Omron CX-Programmer project New_Project (CX-Programmer 9.73)

# PLC NewPLC1: CP2E-N N

## Global symbols (name address type ; comment)
ModbusServer _CP2E003_ExecuteModTcpServer

## Program New_Program1 (cyclic task 0)

### Section Section1

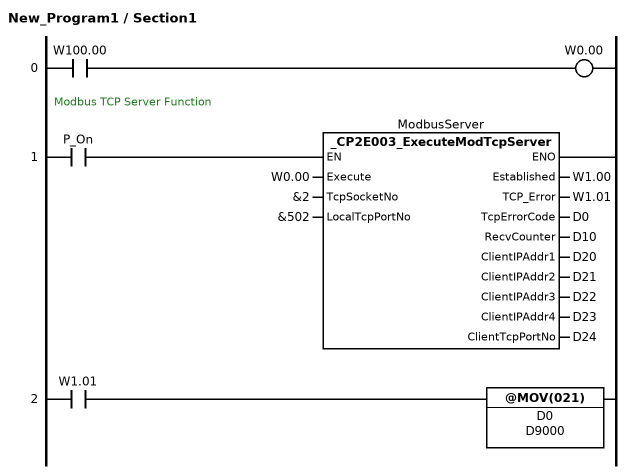
; rung 0
LD W100.00
OUT W0.00
; rung 1: Modbus TCP Server Function
LD P_On
CALL ModbusServer : _CP2E003_ExecuteModTcpServer (Execute := W0.00, TcpSocketNo := &2, LocalTcpPortNo := &502, Established => W1.00, TCP_Error => W1.01, TcpErrorCode => D0, RecvCounter => D10, ClientIPAddr1 => D20, ClientIPAddr2 => D21, ClientIPAddr3 => D22, ClientIPAddr4 => D23, ClientTcpPortNo => D24)
; rung 2
LD W1.01
@MOV(021) D0 D9000

### Section END
; rung 0
END(001)

## Function block _CP2E003_ExecuteModTcpServer (Omron library block, body left out)